FUNCTION_BLOCK skTransfer (* Composite Function Block Type *)
  (* Standard: 61499-2 *)
  (* Version 0.0, 11/8/2025, vv263, template *)
  PACKAGE Main;
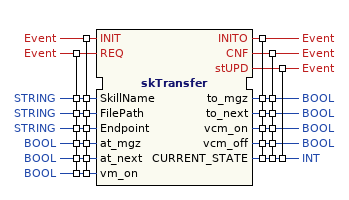
  EVENT_INPUT
    INIT WITH SkillName, FilePath, Endpoint, at_mgz, at_next, vm_on; (* Initialization Request *)
    REQ WITH SkillName, FilePath, Endpoint, at_mgz, at_next, vm_on; (* Normal Execution Request *)
  END_EVENT
  EVENT_OUTPUT
    INITO WITH to_mgz, to_next, CURRENT_STATE, vcm_on, vcm_off; (* Initialization Confirm *)
    CNF WITH to_mgz, to_next, CURRENT_STATE, vcm_on, vcm_off; (* Execution Confirmation *)
    stUPD WITH CURRENT_STATE;
  END_EVENT
  VAR_INPUT
    SkillName : STRING;
    FilePath : STRING;
    Endpoint : STRING;
    at_mgz : BOOL;
    at_next : BOOL;
    vm_on : BOOL;
  END_VAR
  VAR_OUTPUT
    to_mgz : BOOL;
    to_next : BOOL;
    vcm_on : BOOL;
    vcm_off : BOOL;
    CURRENT_STATE : INT;
  END_VAR
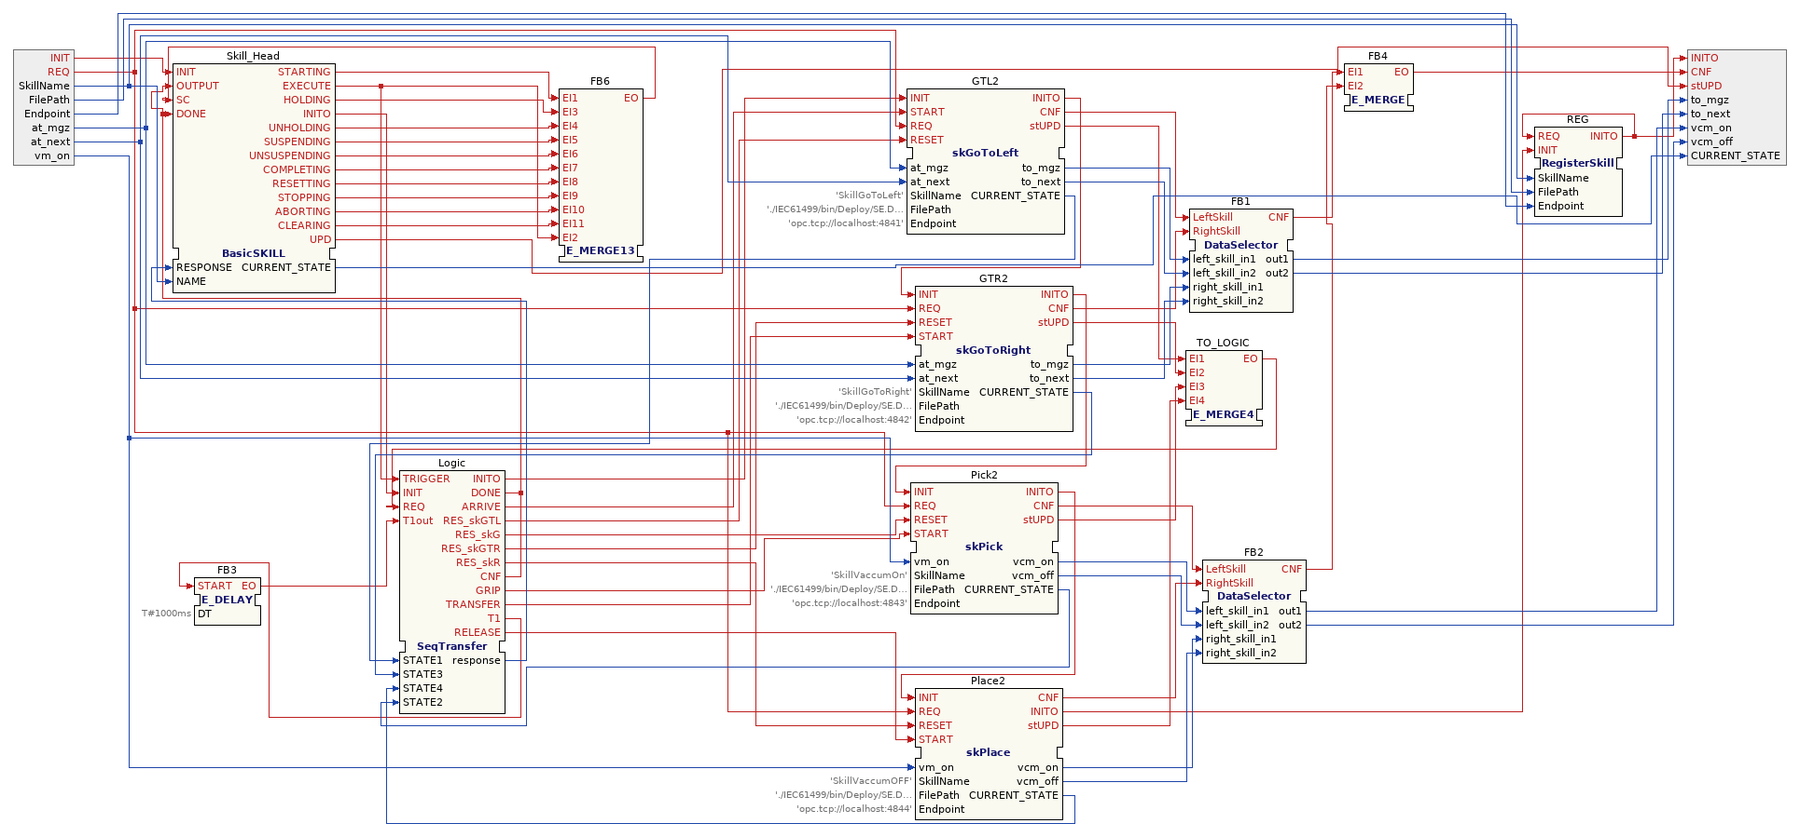
  FBS
    Skill_Head : BasicSKILL;
    REG : RegisterSkill;
    FB1 : DataSelector;
    FB2 : DataSelector;
    GTL2 : skGoToLeft(SkillName := 'SkillGoToLeft', FilePath := './IEC61499/bin/Deploy/SE.DPAC#Soft_dPAC/System.PLC.opcua.xml', Endpoint := 'opc.tcp://localhost:4841');
    GTR2 : skGoToRight(SkillName := 'SkillGoToRight', FilePath := './IEC61499/bin/Deploy/SE.DPAC#Soft_dPAC/System.PLC.opcua.xml', Endpoint := 'opc.tcp://localhost:4842');
    Pick2 : skPick(SkillName := 'SkillVaccumOn', FilePath := './IEC61499/bin/Deploy/SE.DPAC#Soft_dPAC/System.PLC.opcua.xml', Endpoint := 'opc.tcp://localhost:4843');
    Place2 : skPlace(SkillName := 'SkillVaccumOFF', FilePath := './IEC61499/bin/Deploy/SE.DPAC#Soft_dPAC/System.PLC.opcua.xml', Endpoint := 'opc.tcp://localhost:4844');
    Logic : SeqTransfer;
    FB4 : E_MERGE;
    FB6 : E_MERGE13;
    TO_LOGIC : E_MERGE4;
    FB3 : E_DELAY(DT := T#1000ms);
  END_FBS
  EVENT_CONNECTIONS
    Skill_Head.STARTING TO FB6.EI1;
    Skill_Head.EXECUTE TO Logic.TRIGGER;
    Skill_Head.HOLDING TO FB6.EI3;
    INIT TO Skill_Head.INIT;
    Skill_Head.INITO TO Logic.INIT;
    Logic.INITO TO GTL2.INIT;
    REG.INITO TO REG.REQ;
    REG.INITO TO INITO;
    FB4.EO TO CNF;
    Skill_Head.UNHOLDING TO FB6.EI4;
    Skill_Head.SUSPENDING TO FB6.EI5;
    Skill_Head.UNSUSPENDING TO FB6.EI6;
    Skill_Head.COMPLETING TO FB6.EI7;
    Skill_Head.RESETTING TO FB6.EI8;
    Skill_Head.STOPPING TO FB6.EI9;
    Skill_Head.ABORTING TO FB6.EI10;
    Skill_Head.CLEARING TO FB6.EI11;
    Logic.DONE TO Skill_Head.OUTPUT;
    GTL2.INITO TO GTR2.INIT;
    GTR2.INITO TO Pick2.INIT;
    Pick2.INITO TO Place2.INIT;
    GTL2.CNF TO FB1.LeftSkill;
    GTR2.CNF TO FB1.RightSkill;
    Pick2.CNF TO FB2.LeftSkill;
    Place2.CNF TO FB2.RightSkill;
    FB1.CNF TO FB4.EI1;
    FB2.CNF TO FB4.EI2;
    GTL2.stUPD TO TO_LOGIC.EI1;
    Place2.INITO TO REG.INIT;
    Logic.ARRIVE TO GTL2.START;
    REQ TO GTL2.REQ;
    REQ TO GTR2.REQ;
    REQ TO Pick2.REQ;
    REQ TO Place2.REQ;
    FB6.EO TO Skill_Head.SC;
    Logic.DONE TO Skill_Head.DONE;
    GTR2.stUPD TO TO_LOGIC.EI2;
    Pick2.stUPD TO TO_LOGIC.EI3;
    Place2.stUPD TO TO_LOGIC.EI4;
    TO_LOGIC.EO TO Logic.REQ;
    Logic.RES_skGTL TO GTL2.RESET;
    Logic.RES_skG TO Pick2.RESET;
    Logic.RES_skGTR TO GTR2.RESET;
    Logic.RES_skR TO Place2.RESET;
    Skill_Head.UPD TO stUPD;
    Logic.CNF TO Skill_Head.OUTPUT;
    Logic.GRIP TO Pick2.START;
    Logic.TRANSFER TO GTR2.START;
    Logic.T1 TO FB3.START;
    FB3.EO TO Logic.T1out;
    Logic.RELEASE TO Place2.START;
    Skill_Head.EXECUTE TO FB6.EI2;
  END_CONNECTIONS
  DATA_CONNECTIONS
    SkillName TO REG.SkillName;
    FilePath TO REG.FilePath;
    Endpoint TO REG.Endpoint;
    at_mgz TO GTL2.at_mgz;
    at_next TO GTL2.at_next;
    FB1.out1 TO to_mgz;
    FB1.out2 TO to_next;
    Logic.response TO Skill_Head.RESPONSE;
    SkillName TO Skill_Head.NAME;
    GTL2.to_mgz TO FB1.left_skill_in1;
    GTL2.to_next TO FB1.left_skill_in2;
    GTR2.to_mgz TO FB1.right_skill_in1;
    GTR2.to_next TO FB1.right_skill_in2;
    Pick2.vcm_on TO FB2.left_skill_in1;
    Pick2.vcm_off TO FB2.left_skill_in2;
    Place2.vcm_on TO FB2.right_skill_in1;
    Place2.vcm_off TO FB2.right_skill_in2;
    at_mgz TO GTR2.at_mgz;
    at_next TO GTR2.at_next;
    Skill_Head.CURRENT_STATE TO CURRENT_STATE;
    vm_on TO Pick2.vm_on;
    vm_on TO Place2.vm_on;
    FB2.out1 TO vcm_on;
    FB2.out2 TO vcm_off;
    GTL2.CURRENT_STATE TO Logic.STATE1;
    GTR2.CURRENT_STATE TO Logic.STATE3;
    Place2.CURRENT_STATE TO Logic.STATE4;
    Pick2.CURRENT_STATE TO Logic.STATE2;
  END_CONNECTIONS
END_FUNCTION_BLOCK
